(* CODESYS project Modbus.project

Project tree, tasks and I/O mapping:
  Device : AC801-0221-U0R0, Shenzhen Inovance Technology Co., Ltd., version 3.5.11.50
    application Application
      libraries: Standard, * (System)
      task MainTask (cyclic, interval 4 ms, priority 2) calls PLC_PRG
      program PLC_PRG [ST]
      DifferentialMonitor
    HardWare Configuration
    Network Configuration
    Device Diagnosis
    Resources List
    ConfigStorage
    SoftMotion General Axis Pool
    HwConfiguratioinDevice : SystemConfig, Inovance, version 00.00.00.10
        settings: NetworkConfigArray.NetworkConfigArray.BusType = 10; NetworkConfigArray.NetworkConfigArray.RackSum = 1; NetworkConfigArray.NetworkConfigArray.HardwareConfigArray.HardwareConfigArray.RackNo = 1; EnableFun = 12
    MODBUS_COM1 : Modbus主站, inovance, version 00.00.00.10
        settings: Vendor.parameterset.Bit0 = True; Vendor.parameterset.Bit1 = False; Vendor.parameterset.Bit2 = True; Vendor.parameterset.Bit3 = False; Vendor.parameterset.Bit6 = False; Vendor.parameterset.Bit7 = False; modbus master com port.SlaveNum = 1; modbus master com port.FrameDelay = 10;  = 1; IsVirtual = False
      modbus_protocol : Modbus Slave, Inovance, version 00.00.00.10
          settings: UseDec = False; modbus slave com port.ChannelNum = 10; modbus slave com port.ModbusComSet = 1; modbus slave com port.EnableSlaveVariable = 2001; channel.PremeterSet.Bit3 = TRUE; channel.CycleTimes = 200; channel.ReadRegOffSet = 45056; channel.ReadRegLeg = 28; channel.WriteRegOffSet = 0; channel.IOChannel = 0; channel.ResendCount = 1; channel.ChannelName = 'BMS数据'; channel.ChannelNote = ''; channel.PremeterSet.Bit3 = TRUE; channel.CycleTimes = 200; channel.ReadRegOffSet = 4352; channel.ReadRegLeg = 30; channel.WriteRegOffSet = 0; channel.ResendCount = 1; channel.ChannelName = '电池反馈数据组1'; channel.ChannelNote = ''; channel.PremeterSet.Bit3 = TRUE; channel.CycleTimes = 200; channel.ReadRegOffSet = 4416; channel.ReadRegLeg = 30; channel.WriteRegOffSet = 0; channel.IOChannel = 2; channel.ResendCount = 1; channel.ChannelName = '电池反馈数据组2'; channel.ChannelNote = ''; channel.PremeterSet.Bit3 = TRUE; channel.CycleTimes = 200; channel.ReadRegOffSet = 4480; channel.ReadRegLeg = 30; channel.WriteRegOffSet = 0; channel.IOChannel = 3; channel.ResendCount = 1; channel.ChannelName = '电池反馈数据组3'; channel.ChannelNote = ''; channel.PremeterSet.Bit3 = TRUE;
            channel.CycleTimes = 200; channel.ReadRegOffSet = 4544; channel.ReadRegLeg = 30; channel.WriteRegOffSet = 0; channel.IOChannel = 4; channel.ResendCount = 1; channel.ChannelName = '电池反馈数据组4'; channel.ChannelNote = ''; channel.PremeterSet.Bit3 = TRUE; channel.CycleTimes = 200; channel.ReadRegOffSet = 16640; channel.ReadRegLeg = 10; channel.WriteRegOffSet = 0; channel.IOChannel = 5; channel.ResendCount = 1; channel.ChannelName = '电池温度组1'; channel.ChannelNote = ''; channel.PremeterSet.Bit3 = TRUE; channel.CycleTimes = 200; channel.ReadRegOffSet = 16706; channel.ReadRegLeg = 10; channel.WriteRegOffSet = 0; channel.IOChannel = 6; channel.ResendCount = 1; channel.ChannelName = '电池温度组2'; channel.ChannelNote = ''; channel.PremeterSet.Bit3 = TRUE; channel.CycleTimes = 200; channel.ReadRegOffSet = 16772; channel.ReadRegLeg = 10; channel.WriteRegOffSet = 0; channel.IOChannel = 7; channel.ResendCount = 1; channel.ChannelName = '电池温度组3'; channel.ChannelNote = ''; channel.PremeterSet.Bit3 = TRUE; channel.CycleTimes = 200; channel.ReadRegOffSet = 16838; channel.ReadRegLeg = 10; channel.WriteRegOffSet = 0;
            channel.IOChannel = 8; channel.ResendCount = 1; channel.ChannelName = '电池温度组4'; channel.ChannelNote = ''; channel.PremeterSet.Bit3 = TRUE; channel.CycleTimes = 200; channel.ReadRegOffSet = 40960; channel.ReadRegLeg = 27; channel.WriteRegOffSet = 0; channel.IOChannel = 9; channel.ResendCount = 1; channel.ChannelName = 'UPS反馈数据'; channel.ChannelNote = ''
          input  Application.PLC_PRG.BMS映射数据 AT %IW0 :  ARRAY[0..27] OF WORD  // BMS数据
          input  Application.PLC_PRG.电池映射电压组1 :  ARRAY[0..29] OF WORD  // 电池反馈数据组1
          input  Application.PLC_PRG.电池映射电压组2 :  ARRAY[0..29] OF WORD  // 电池反馈数据组2
          input  Application.PLC_PRG.电池映射电压组3 :  ARRAY[0..29] OF WORD  // 电池反馈数据组3
          input  Application.PLC_PRG.电池映射电压组4 :  ARRAY[0..29] OF WORD  // 电池反馈数据组4
          input  Application.PLC_PRG.电池映射温度组1 :  ARRAY[0..9] OF WORD  // 电池温度组1
          input  Application.PLC_PRG.电池映射温度组2 :  ARRAY[0..9] OF WORD  // 电池温度组2
          input  Application.PLC_PRG.电池映射温度组3 :  ARRAY[0..9] OF WORD  // 电池温度组3
          input  Application.PLC_PRG.电池映射温度组4 :  ARRAY[0..9] OF WORD  // 电池温度组4
          input  Application.PLC_PRG.UPS映射数据 :  ARRAY[0..26] OF WORD  // UPS反馈数据
    MODBUS_TCP_1 : ModbusTCP主站, inovance, version 00.00.00.10
        settings: ModbusTcpMaster.SlaveNUm = 0;  = 0
*)

// Device/Application/PLC_PRG
PROGRAM PLC_PRG
VAR
	BMS映射数据 : ARRAY [0..27] OF WORD; // 16位数组
	UPS映射数据 : ARRAY [0..26] OF WORD; // 0x3030为正常状态
	电池映射电压组1 : ARRAY [0..29] OF WORD;
	电池映射电压组2 : ARRAY [0..29] OF WORD;
	电池映射电压组3 : ARRAY [0..29] OF WORD;
	电池映射电压组4 : ARRAY [0..29] OF WORD;
	电池映射温度组1 : ARRAY [0..9] OF WORD;
	电池映射温度组2 : ARRAY [0..9] OF WORD;
	电池映射温度组3 : ARRAY [0..9] OF WORD;
	电池映射温度组4 : ARRAY [0..9] OF WORD;
	
	iCounter : INT := 0;
	系统状态 : INT := 0;
	电池状态 : INT := 0;
	一级保护状态 : DWORD := 0;
	二级保护状态 : DWORD := 0;
	三级保护状态 : DWORD := 0;
	故障状态 : DWORD := 0;
	采集电压 : LREAL := 0.0;
	负载电压 : LREAL := 0.0;
	上桥累计电压 : LREAL := 0.0;
	下桥累计电压 : LREAL := 0.0;
	上桥电流 : LREAL := 0.0;
	下桥电流 : LREAL := 0.0;
	上桥SOC : LREAL := 0.0;
	下桥SOC : LREAL := 0.0;
	上桥SOH : LREAL := 0.0;
	下桥SOH : LREAL := 0.0;
	上桥电池剩余容量 : LREAL := 0.0;
	下桥电池剩余容量 : LREAL := 0.0;
	上桥系统功率 : LREAL := 0.0;
	下桥系统功率 : LREAL := 0.0;
	
	UPS警告项1 : WORD := 0;
	UPS警告项2 : WORD := 0;
	UPS警告项3 : WORD := 0;
	UPS警告项4 : WORD := 0;
	UPS警告项5 : WORD := 0;
	R输入电压 : LREAL := 0.0;
	S输入电压 : LREAL := 0.0;
	T输入电压 : LREAL := 0.0;
	R输出电压 : LREAL := 0.0;
	S输出电压 : LREAL := 0.0;
	T输出电压 : LREAL := 0.0;
	输出频率 : LREAL := 0.0;
	R输出电流 : LREAL := 0.0;
	S输出电流 : LREAL := 0.0;
	T输出电流 : LREAL := 0.0;
	R输出负载百分比 : LREAL := 0.0;
	S输出负载百分比 : LREAL := 0.0;
	T输出负载百分比 : LREAL := 0.0;
	总输出负载百分比 : LREAL := 0.0;
	UPS状态 : WORD := 0;
	散热器温度1 : LREAL := 0.0;
	散热器温度2 : LREAL := 0.0;
	机柜温度 : LREAL := 0.0;
	UPS模式 : WORD := 0;
	UPS故障信息 : WORD := 0;			
	当前功率 : LREAL := 0.0;

	电池反馈电压组1 : ARRAY [0..29] OF LREAL;
	电池反馈电压组2 : ARRAY [0..29] OF LREAL;
	电池反馈电压组3 : ARRAY [0..29] OF LREAL;
	电池反馈电压组4 : ARRAY [0..29] OF LREAL;
	电池反馈温度组1 : ARRAY [0..9] OF LREAL;
	电池反馈温度组2 : ARRAY [0..9] OF LREAL;
	电池反馈温度组3 : ARRAY [0..9] OF LREAL;
	电池反馈温度组4 : ARRAY [0..9] OF LREAL;
	
	// ARR0 AT %MW0: ARRAY [0..9] OF WORD :=[0,2,4,6,8,10,1,3,5,7];
END_VAR

系统状态 := WORD_TO_INT(BMS映射数据[0]); // 0-初始化 1-待机模式 2-充电模式 3-放电模式 4-上电BCU编码中 5-上电BMU编码中 6-上电绝缘检测中 7-上电并机中 8-掉电中 9-系统锁定
电池状态 := WORD_TO_INT(BMS映射数据[1]); // 0-等待 1-禁充禁放 2-禁充 3-禁放 4-充电中 5-放电中
一级保护状态 := SHL(BMS映射数据[2], 16) OR BMS映射数据[3];
二级保护状态 := SHL(BMS映射数据[4], 16) OR BMS映射数据[5];
三级保护状态 := SHL(BMS映射数据[6], 16) OR BMS映射数据[7];
故障状态 := SHL(BMS映射数据[8], 16) OR BMS映射数据[9];
采集电压 := WORD_TO_LREAL(BMS映射数据[10]) * 0.1; 		// 转换为V
负载电压 := WORD_TO_LREAL(BMS映射数据[11]) * 0.1; 		// 转换为V
上桥累计电压 := WORD_TO_LREAL(BMS映射数据[12]) * 0.1; 	// 转换为V
下桥累计电压 := WORD_TO_LREAL(BMS映射数据[13]) * 0.1; 	// 转换为V
上桥电流 := DWORD_TO_DINT(SHL(BMS映射数据[14], 16) OR BMS映射数据[15]) * 0.01; // 转换为A
下桥电流 := DWORD_TO_DINT(SHL(BMS映射数据[16], 16) OR BMS映射数据[17]) * 0.01; // 转换为A
上桥SOC := WORD_TO_LREAL(BMS映射数据[18]); // 单位%
下桥SOC := WORD_TO_LREAL(BMS映射数据[19]); // 单位%
上桥SOH := WORD_TO_LREAL(BMS映射数据[20]); // 单位%
下桥SOH := WORD_TO_LREAL(BMS映射数据[21]); // 单位%
上桥电池剩余容量 := DWORD_TO_DINT(SHL(BMS映射数据[22], 16) OR BMS映射数据[23]) * 0.01; // 单位AH
下桥电池剩余容量 := DWORD_TO_DINT(SHL(BMS映射数据[24], 16) OR BMS映射数据[25]) * 0.01; // 单位AH
上桥系统功率 := WORD_TO_LREAL(BMS映射数据[26]) * 0.1; // 单位KW
下桥系统功率 := WORD_TO_LREAL(BMS映射数据[27]) * 0.1; // 单位KW

UPS警告项1 := UPS映射数据[0];
UPS警告项2 := UPS映射数据[1];
UPS警告项3 := UPS映射数据[2];
UPS警告项4 := UPS映射数据[3];
UPS警告项5 := UPS映射数据[4];
R输入电压 := WORD_TO_LREAL(UPS映射数据[5]) * 0.01804; 		// 转换为V
S输入电压 := WORD_TO_LREAL(UPS映射数据[6]) * 0.01804; 		// 转换为V
T输入电压 := WORD_TO_LREAL(UPS映射数据[7]) * 0.01804; 		// 转换为V
R输出电压 := WORD_TO_LREAL(UPS映射数据[9]) * 0.1; 			// 转换为V
S输出电压 := WORD_TO_LREAL(UPS映射数据[10]) * 0.1; 		// 转换为V
T输出电压 := WORD_TO_LREAL(UPS映射数据[11]) * 0.1; 		// 转换为V
输出频率 := WORD_TO_LREAL(UPS映射数据[12]) * 0.1; 			// 转换为Hz
R输出电流 := WORD_TO_LREAL(UPS映射数据[13]) * 0.1; 		// 转换为A
S输出电流 := WORD_TO_LREAL(UPS映射数据[14]) * 0.1; 		// 转换为A
T输出电流 := WORD_TO_LREAL(UPS映射数据[15]) * 0.1; 		// 转换为A
R输出负载百分比 := WORD_TO_LREAL(UPS映射数据[16]) * 0.1; 	// 转换为%
S输出负载百分比 := WORD_TO_LREAL(UPS映射数据[17]) * 0.1; 	// 转换为%
T输出负载百分比 := WORD_TO_LREAL(UPS映射数据[18]) * 0.1; 	// 转换为%
总输出负载百分比 := WORD_TO_LREAL(UPS映射数据[19]) * 0.1; 	// 转换为%
UPS状态 := UPS映射数据[20];
散热器温度1 := WORD_TO_LREAL(UPS映射数据[21]); // 转换为度
散热器温度2 := WORD_TO_LREAL(UPS映射数据[22]); // 转换为度
机柜温度 := WORD_TO_LREAL(UPS映射数据[23]); 	// 转换为度
UPS模式 := UPS映射数据[24]; //0x50-开机模式 0x53-待机模式 0x59-旁路模式 0x4C-线路模式 0x42-电池模式 0x46-故障模式 0x45-HE/ECO模式 0x43-转换器模式 0x44-关机模式 
UPS故障信息 := UPS映射数据[25];
当前功率 := WORD_TO_LREAL(UPS映射数据[26]); 	// 转换为W

FOR iCounter:=0 TO 29 BY 1 DO
	电池反馈电压组1[iCounter] := WORD_TO_LREAL(电池映射电压组1[iCounter]) * 0.001; // 转换为V
	电池反馈电压组2[iCounter] := WORD_TO_LREAL(电池映射电压组2[iCounter]) * 0.001; // 转换为V
	电池反馈电压组3[iCounter] := WORD_TO_LREAL(电池映射电压组3[iCounter]) * 0.001; // 转换为V
	电池反馈电压组4[iCounter] := WORD_TO_LREAL(电池映射电压组4[iCounter]) * 0.001; // 转换为V
END_FOR

FOR iCounter:=0 TO 9 BY 1 DO
	电池反馈温度组1[iCounter] := 电池映射温度组1[iCounter] * 0.1; // 转换为度
	电池反馈温度组2[iCounter] := 电池映射温度组2[iCounter] * 0.1; // 转换为度
	电池反馈温度组3[iCounter] := 电池映射温度组3[iCounter] * 0.1; // 转换为度
	电池反馈温度组4[iCounter] := 电池映射温度组4[iCounter] * 0.1; // 转换为度
END_FOR

END_PROGRAM
